(* Logix 5000 project; controller cal1615 1756-L62 rev 20.11; software revision 20.05; part 13 of 81 *)
(* tags used below, declared in another part *)
   FAULT : BOOL;   // Fault AFI
   p01_ai_prs : REAL;   // System Inputs Oxidizer Differential Pressure
   p01_ai_tc : REAL;   // System Inputs Oxidizer Inlet Temperature
   p01_int_from_oxidizer : INT[10];   // System Oxidizer Int from Oxidizer
   p01_int_to_oxidizer : INT;   // System Oxidizer Int to Oxidizer
   p01_param_tension_deviation : REAL;
   p01r01 : routine;
   p01r03_oxidizer_prs : SYS_SCP;   // System Inputs Oxidizer Differential Pressure Scaling
   p01r03_prs_input_max : REAL;
   p01r03_prs_input_min : REAL;
   p01r03_prs_output_max : REAL;
   p01r03_prs_output_min : REAL;
   p01r09_pb_global_reset : BOOL;   // System Modes PB: Global Fault Reset
   p01r12_master_ramped_speed : REAL;   // System Line Accel Decel Control Master Ramped Speed
   p01r12_selected_line_speed : REAL;   // System Line Accel Decel Control Selected Line Speed
   p01r13 : routine;   // System Line Start Sequence
   p01r13_check_status : BOOL;   // System Line Start Sequence Check Status
   p01r13_check_status_time : REAL;   // System Line Start Sequence Check Status
   p01r13_check_status_timer : TIMER;   // System Line Start Sequence Check Status Timer
   p01r13_check_tension : TIMER;   // System Line Start Sequence Check Tension
   p01r13_letoff_tension_ok : BOOL;   // System Line Start Sequence Letoff Tension Ok
   p01r13_line_running : BOOL;   // System Line Start Sequence Line Running
   p01r13_line_slow_ramp : BOOL;   // System Line Start Sequence Start Line to Slow Speed
   p01r13_line_start : SYS_ENC;   // System Line Start Sequence Encoder
   p01r13_permissive_drives : BOOL;   // System Line Start Sequence Permissive Drives
   p01r13_permissive_line_run : BOOL;   // System Line Start Sequence Permissive Line Run
   p01r13_permissive_oven : BOOL;   // System Line start Sequence Permissive Ovens
   p01r13_request_run : BOOL;   // System Line Start Sequence Request Run
   p01r13_request_stop : BOOL;   // System Line Start Sequence Request Stop
   p01r13_state : DINT;   // System Line Start Sequence Sequencer Step
   p01r13_status : DINT;   // System Line Start Sequence Encoded Step
   p01r13_tension_ok : BOOL;   // System Line Start Sequence Slow Speed Tension Ok
   p01r13_timer_fault : TIMER[8];   // System Line Start Sequence Fault Dwell Timer
   p01r13_timer_line_start_warning_dwell : TIMER;   // System Line Start Sequence Pre Start Warning Dwell Timer
   p01r13_timer_line_stop_dwell : TIMER;   // System Line Start Sequence Line Stop Dwell Timer
   p01r13_timer_switch_to_stretch_dwell : TIMER;   // System Line Start Sequence Setpoint Stretch to Tension Dwell Timer
   p01r13_timer_warning : TIMER[8];   // System Line Start Sequence Warning Dwell Timer
   p01r13_ts1_tension_ok : BOOL;   // System Line Start Sequence TS 1 Tension Ok
   p01r13_ts2_tension_ok : BOOL;   // System Line Start Sequence TS 2 Tension Ok
   p01r13_winder_tension_ok : BOOL;   // System Line Start Sequence Winder Tension Ok
   p01r14 : routine;
   p01r14_msg_read : MESSAGE;   // System Oxidizer Message Read
   p01r14_msg_read_retry_timer : TIMER;
   p01r14_msg_read_timer : TIMER;   // System Oxidizer Read Dwell
   p01r14_msg_write : MESSAGE;   // System Oxidizer Message Write
   p01r14_msg_write_retry_timer : TIMER;   // System Oxidizer Message Retry Timer
   p01r14_msg_write_timer : TIMER;   // System Oxidizer Message Read Dwell
   p01r14_oxidizer_heart_beat_off : TIMER;   // System Oxidizer Heart Beat Off Timer
   p01r14_oxidizer_heart_beat_ok : BOOL;   // System Oxidizer Heart Beat Ok
   p01r14_oxidizer_heart_beat_on : TIMER;   // System Oxidizer Heart Beat On Timer
   p01r14_oxidizer_mass_flow : REAL;   // System Oxidizer Oxidizer Mass Flow [SCFM]
   p01r14_timer_fault : TIMER[10];   // System Oxidizer Fault Dwell Timer
   p01r14_timer_warning : TIMER[5];
   p11r02_shutdown_temp : BOOL;   // Zone 1 Misc Control Safe Shutdown Temperature
   p11r20_state : DINT;   // Zone 1 Temperature Control State
   p11r30_request_heat : BOOL;   // Zone 1 Temperature Control Request Heat
   p12r02_shutdown_temp : BOOL;   // Zone 2 Misc Control Safe Shutdown Temperature
   p12r20_state : DINT;   // Zone 2 Temperature Control State
   p12r30_request_heat : BOOL;   // Zone 2 Temperature Control Request Heat
   p13r02_shutdown_temp : BOOL;   // Zone 3 Misc Control Safe Shutdown Temperature
   p13r20_state : DINT;   // Zone 3 Temperature Control State
   p13r30_request_cool : BOOL;   // Zone 3 Temperature Control Request Cooling
   p20_di_acc_empty : BOOL;   // Letoff Digital Input Letoff Accumulator Empty Position
   p20r10_pid_tens : PID;   // Letoff Letoff Speed Control Tension PID
   p22r10_pid_psn : PID;   // Tension Stand 1 Speed Tension PID Dancer Position
   p25r10_pid_psn : PID;   // Tension Stand 2 Speed Tension PID Dancer Position Process Variable
   p29r10_tension_error : REAL;   // Winder Winder A Tension Error winder_tension_sp - Load Cell [lbf]
(* P01_System, continued *)

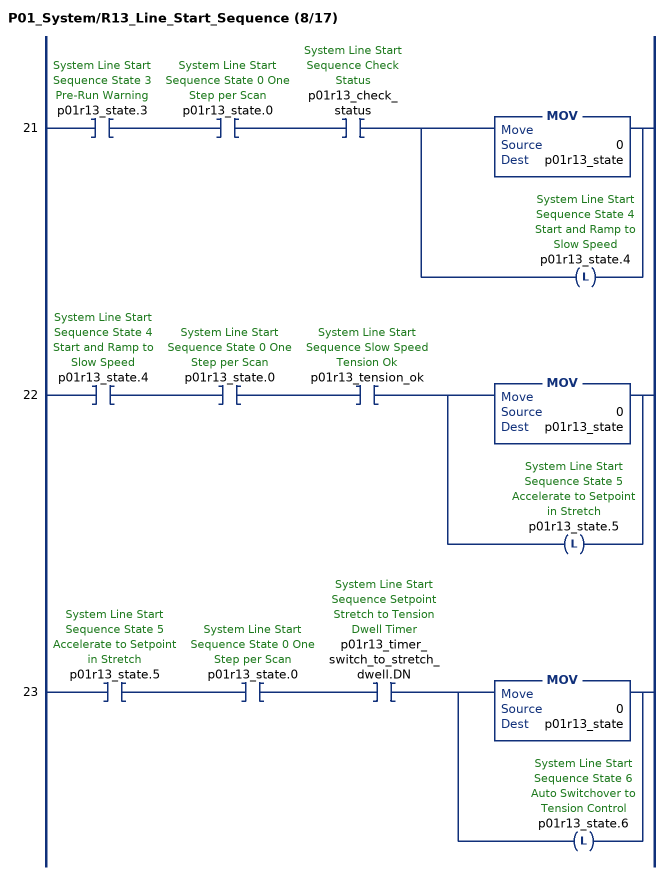
   [picture p162: P01_System/R13_Line_Start_Sequence rungs 21-23]
   21: XIC(p01r13_state.3)XIC(p01r13_state.0)XIC(p01r13_check_status)[MOV(0,p01r13_state) ,OTL(p01r13_state.4) ];
   22: XIC(p01r13_state.4)XIC(p01r13_state.0)XIC(p01r13_tension_ok)[MOV(0,p01r13_state) ,OTL(p01r13_state.5) ];
   23: XIC(p01r13_state.5)XIC(p01r13_state.0)XIC(p01r13_timer_switch_to_stretch_dwell.DN)[MOV(0,p01r13_state) ,OTL(p01r13_state.6) ];
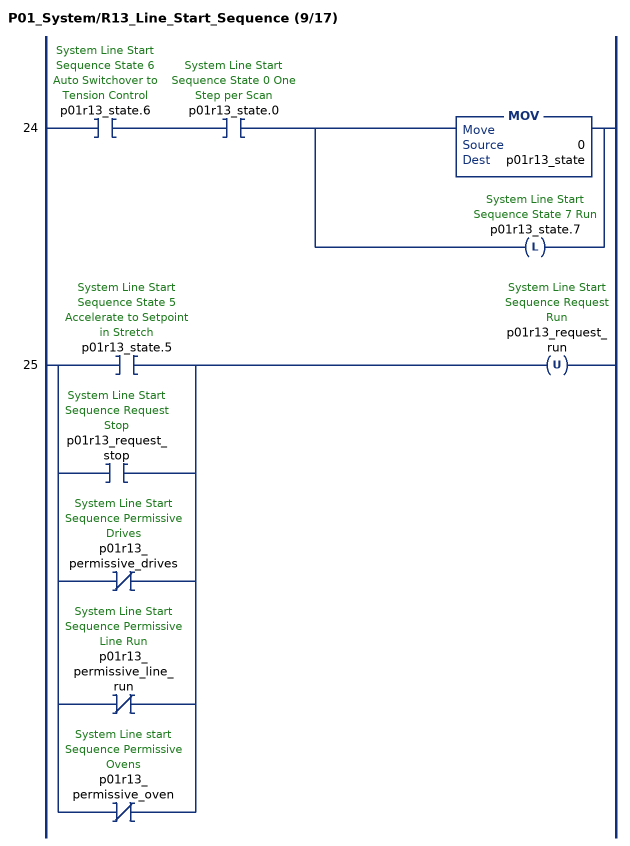
   24: XIC(p01r13_state.6)XIC(p01r13_state.0)[MOV(0,p01r13_state) ,OTL(p01r13_state.7) ];
   25: [XIC(p01r13_state.5) ,XIC(p01r13_request_stop) ,XIO(p01r13_permissive_drives) ,XIO(p01r13_permissive_line_run) ,XIO(p01r13_permissive_oven) ]OTU(p01r13_request_run);
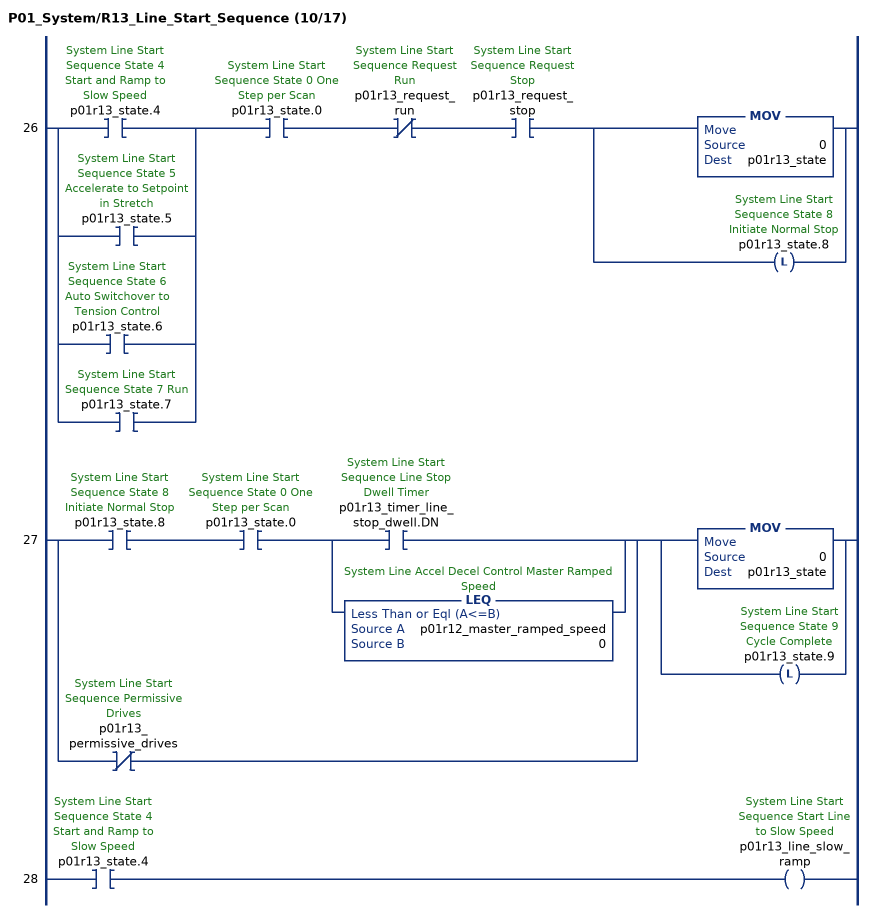
   26: [XIC(p01r13_state.4) ,XIC(p01r13_state.5) ,XIC(p01r13_state.6) ,XIC(p01r13_state.7) ]XIC(p01r13_state.0)XIO(p01r13_request_run)XIC(p01r13_request_stop)[MOV(0,p01r13_state) ,OTL(p01r13_state.8) ];
   27: [XIC(p01r13_state.8) XIC(p01r13_state.0) [XIC(p01r13_timer_line_stop_dwell.DN) ,LEQ(p01r12_master_ramped_speed,0) ] ,XIO(p01r13_permissive_drives) ][MOV(0,p01r13_state) ,OTL(p01r13_state.9) ];
   28: XIC(p01r13_state.4)OTE(p01r13_line_slow_ramp);
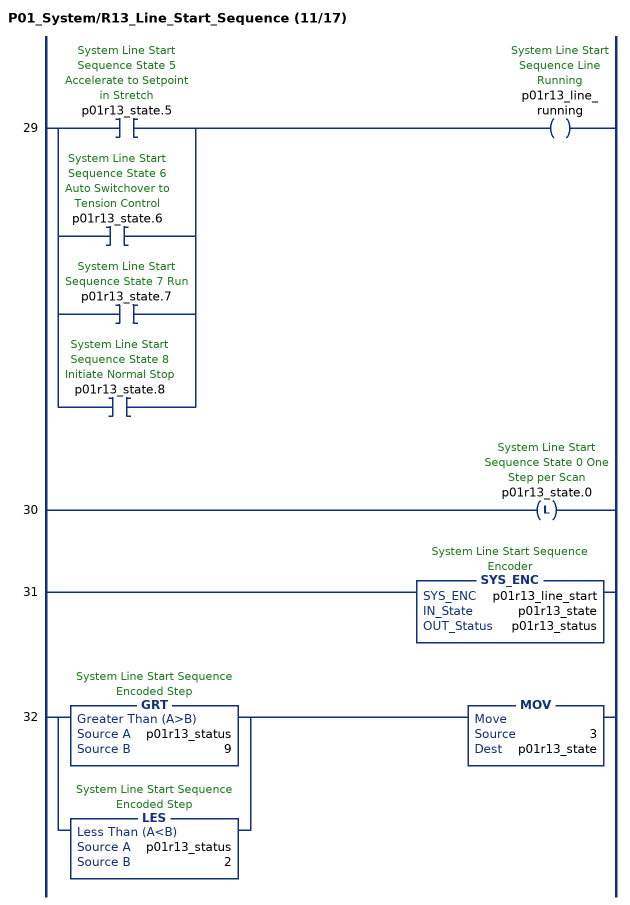
   29: [XIC(p01r13_state.5) ,XIC(p01r13_state.6) ,XIC(p01r13_state.7) ,XIC(p01r13_state.8) ]OTE(p01r13_line_running);
   30: OTL(p01r13_state.0);
   31: SYS_ENC(p01r13_line_start,p01r13_state,p01r13_status);
   32: [GRT(p01r13_status,9) ,LES(p01r13_status,2) ]MOV(3,p01r13_state);
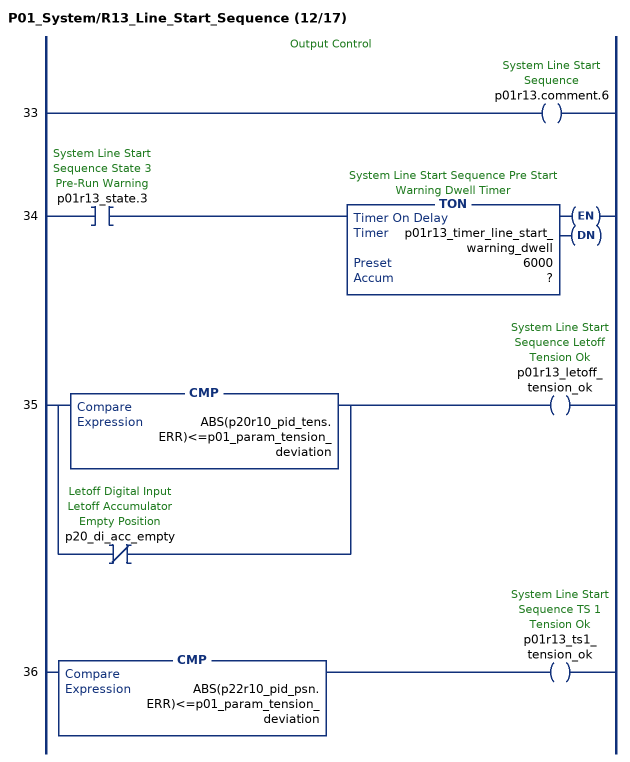
   // Output Control
   33: OTE(p01r13.comment.6);
   34: XIC(p01r13_state.3)TON(p01r13_timer_line_start_warning_dwell,?,?);
   35: [CMP(ABS(p20r10_pid_tens.ERR)<=p01_param_tension_deviation) ,XIO(p20_di_acc_empty) ]OTE(p01r13_letoff_tension_ok);
   36: CMP(ABS(p22r10_pid_psn.ERR)<=p01_param_tension_deviation)OTE(p01r13_ts1_tension_ok);
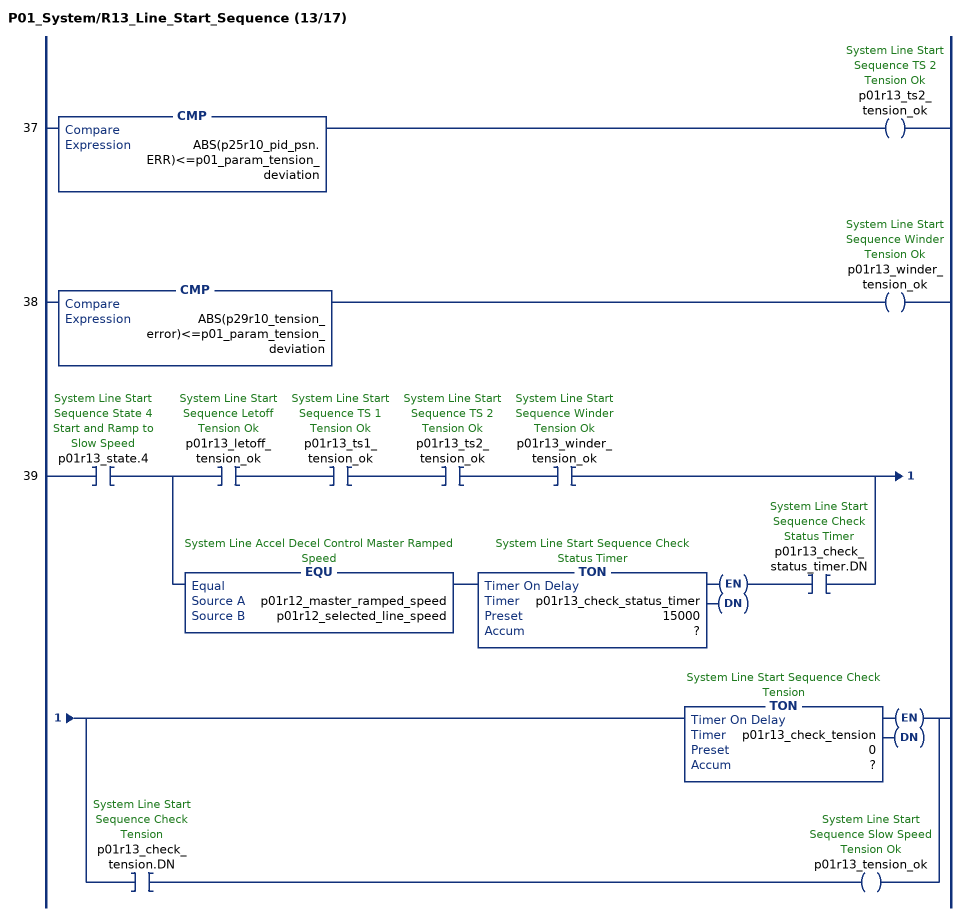
   37: CMP(ABS(p25r10_pid_psn.ERR)<=p01_param_tension_deviation)OTE(p01r13_ts2_tension_ok);
   38: CMP(ABS(p29r10_tension_error)<=p01_param_tension_deviation)OTE(p01r13_winder_tension_ok);
   39: XIC(p01r13_state.4)[XIC(p01r13_letoff_tension_ok) XIC(p01r13_ts1_tension_ok) XIC(p01r13_ts2_tension_ok) XIC(p01r13_winder_tension_ok) ,EQU(p01r12_master_ramped_speed,p01r12_selected_line_speed) TON(p01r13_check_status_timer,?,?) XIC(p01r13_check_status_timer.DN) ][TON(p01r13_check_tension,?,?) ,XIC(p01r13_check_tension.DN) OTE(p01r13_tension_ok) ];
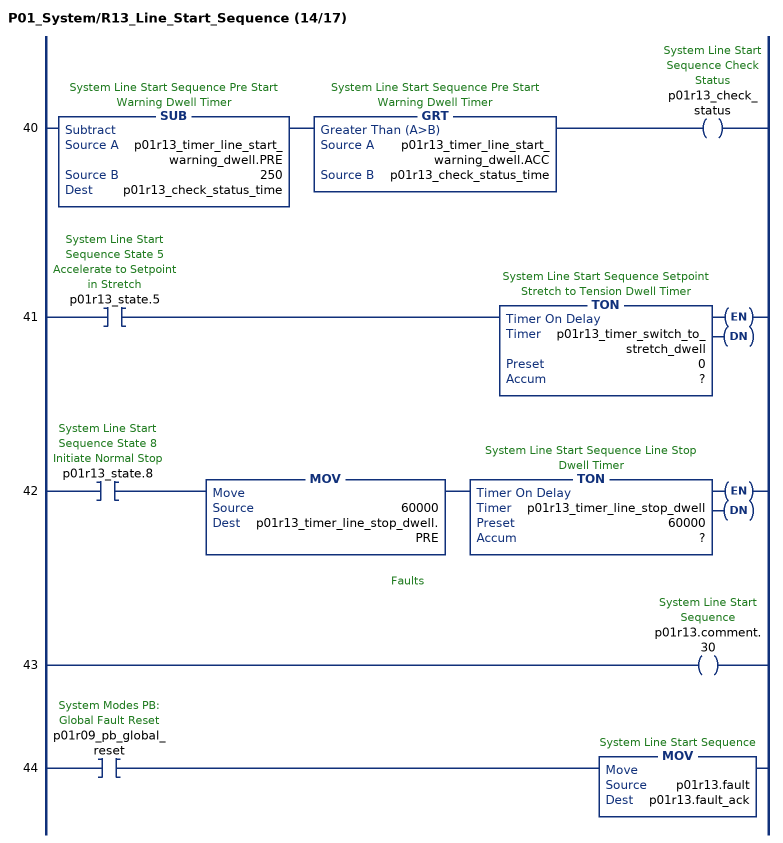
   40: SUB(p01r13_timer_line_start_warning_dwell.PRE,250,p01r13_check_status_time)GRT(p01r13_timer_line_start_warning_dwell.ACC,p01r13_check_status_time)OTE(p01r13_check_status);
   41: XIC(p01r13_state.5)TON(p01r13_timer_switch_to_stretch_dwell,?,?);
   42: XIC(p01r13_state.8)MOV(60000,p01r13_timer_line_stop_dwell.PRE)TON(p01r13_timer_line_stop_dwell,?,?);
   // Faults
   43: OTE(p01r13.comment.30);
   44: XIC(p01r09_pb_global_reset)MOV(p01r13.fault,p01r13.fault_ack);
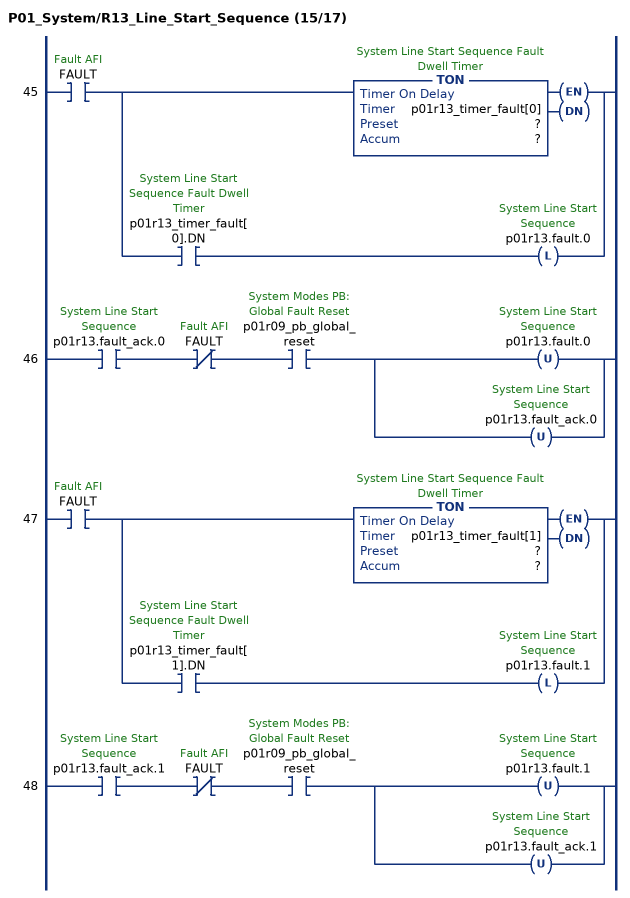
   45: XIC(FAULT)[TON(p01r13_timer_fault[0],?,?) ,XIC(p01r13_timer_fault[0].DN) OTL(p01r13.fault.0) ];
   46: XIC(p01r13.fault_ack.0)XIO(FAULT)XIC(p01r09_pb_global_reset)[OTU(p01r13.fault.0) ,OTU(p01r13.fault_ack.0) ];
   47: XIC(FAULT)[TON(p01r13_timer_fault[1],?,?) ,XIC(p01r13_timer_fault[1].DN) OTL(p01r13.fault.1) ];
   48: XIC(p01r13.fault_ack.1)XIO(FAULT)XIC(p01r09_pb_global_reset)[OTU(p01r13.fault.1) ,OTU(p01r13.fault_ack.1) ];
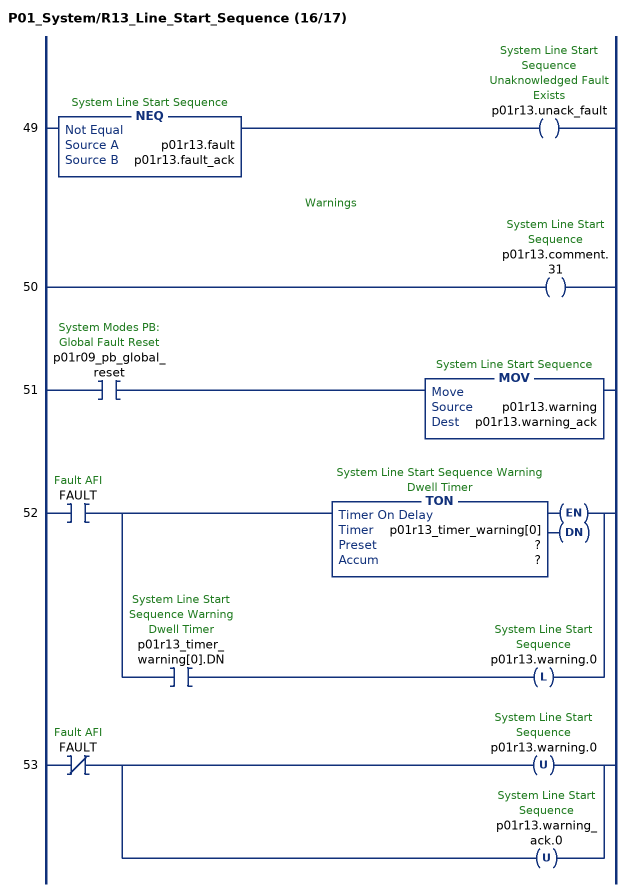
   49: NEQ(p01r13.fault,p01r13.fault_ack)OTE(p01r13.unack_fault);
   // Warnings
   50: OTE(p01r13.comment.31);
   51: XIC(p01r09_pb_global_reset)MOV(p01r13.warning,p01r13.warning_ack);
   52: XIC(FAULT)[TON(p01r13_timer_warning[0],?,?) ,XIC(p01r13_timer_warning[0].DN) OTL(p01r13.warning.0) ];
   53: XIO(FAULT)[OTU(p01r13.warning.0) ,OTU(p01r13.warning_ack.0) ];
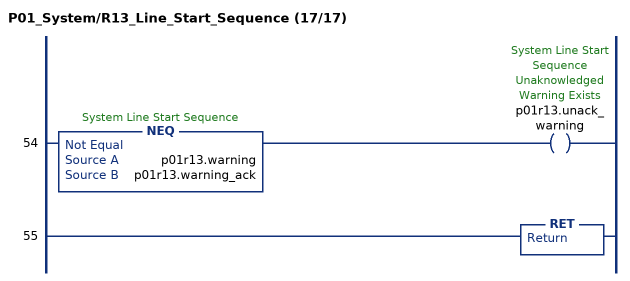
   54: NEQ(p01r13.warning,p01r13.warning_ack)OTE(p01r13.unack_warning);
   55: RET();
END_ROUTINE

ROUTINE R14_Oxidizer   (* ladder *)
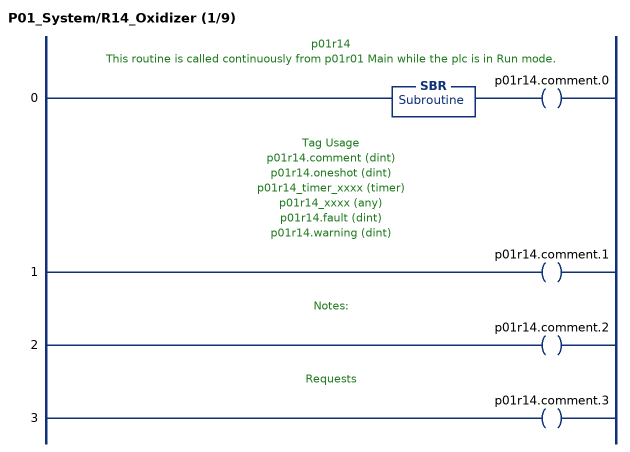
   // p01r14
   // This routine is called continuously from p01r01 Main while the plc is in Run mode.
   0: SBR()OTE(p01r14.comment.0);
   // Tag Usage
   // p01r14.comment (dint)
   // p01r14.oneshot (dint)
   // p01r14_timer_xxxx (timer)
   // p01r14_xxxx (any)
   // p01r14.fault (dint)
   // p01r14.warning (dint)
   1: OTE(p01r14.comment.1);
   // Notes:
   2: OTE(p01r14.comment.2);
   // Requests
   3: OTE(p01r14.comment.3);
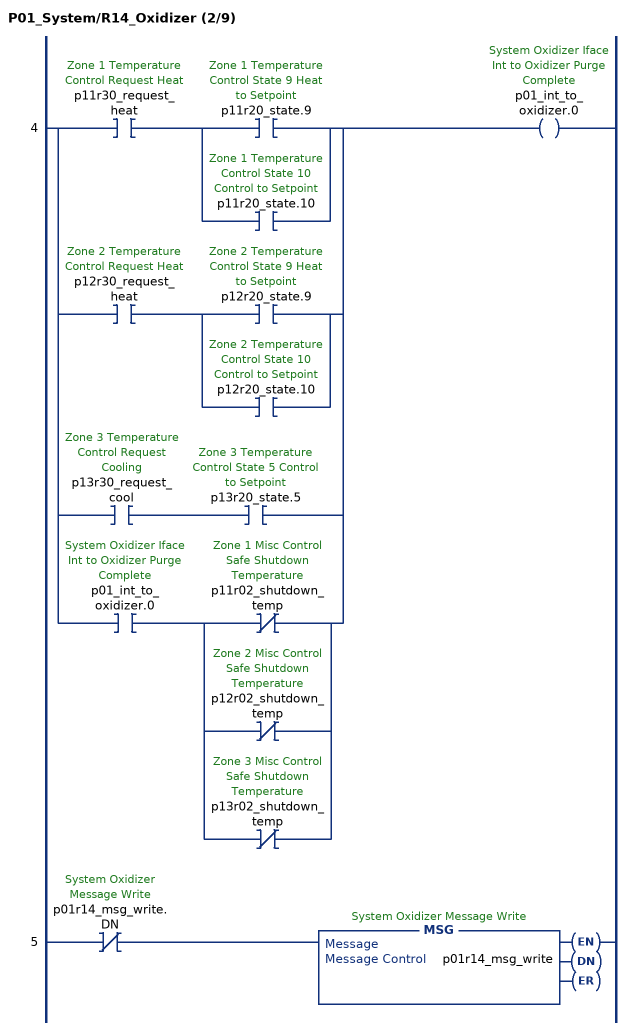
   4: [XIC(p11r30_request_heat) [XIC(p11r20_state.9) ,XIC(p11r20_state.10) ] ,XIC(p12r30_request_heat) [XIC(p12r20_state.9) ,XIC(p12r20_state.10) ] ,XIC(p13r30_request_cool) XIC(p13r20_state.5) ,XIC(p01_int_to_oxidizer.0) [XIO(p11r02_shutdown_temp) ,XIO(p12r02_shutdown_temp) ,XIO(p13r02_shutdown_temp) ] ]OTE(p01_int_to_oxidizer.0);
   5: XIO(p01r14_msg_write.DN)MSG(p01r14_msg_write);
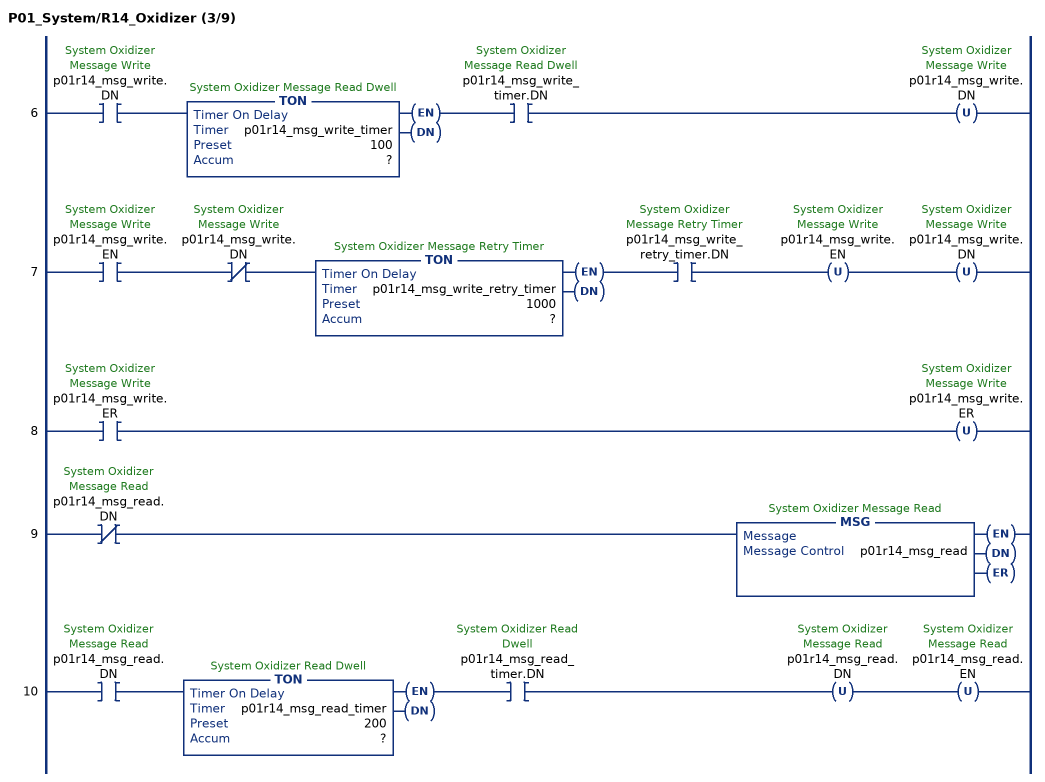
   6: XIC(p01r14_msg_write.DN)TON(p01r14_msg_write_timer,?,?)XIC(p01r14_msg_write_timer.DN)OTU(p01r14_msg_write.DN);
   7: XIC(p01r14_msg_write.EN)XIO(p01r14_msg_write.DN)TON(p01r14_msg_write_retry_timer,?,?)XIC(p01r14_msg_write_retry_timer.DN)OTU(p01r14_msg_write.EN)OTU(p01r14_msg_write.DN);
   8: XIC(p01r14_msg_write.ER)OTU(p01r14_msg_write.ER);
   9: XIO(p01r14_msg_read.DN)MSG(p01r14_msg_read);
   10: XIC(p01r14_msg_read.DN)TON(p01r14_msg_read_timer,?,?)XIC(p01r14_msg_read_timer.DN)OTU(p01r14_msg_read.DN)OTU(p01r14_msg_read.EN);
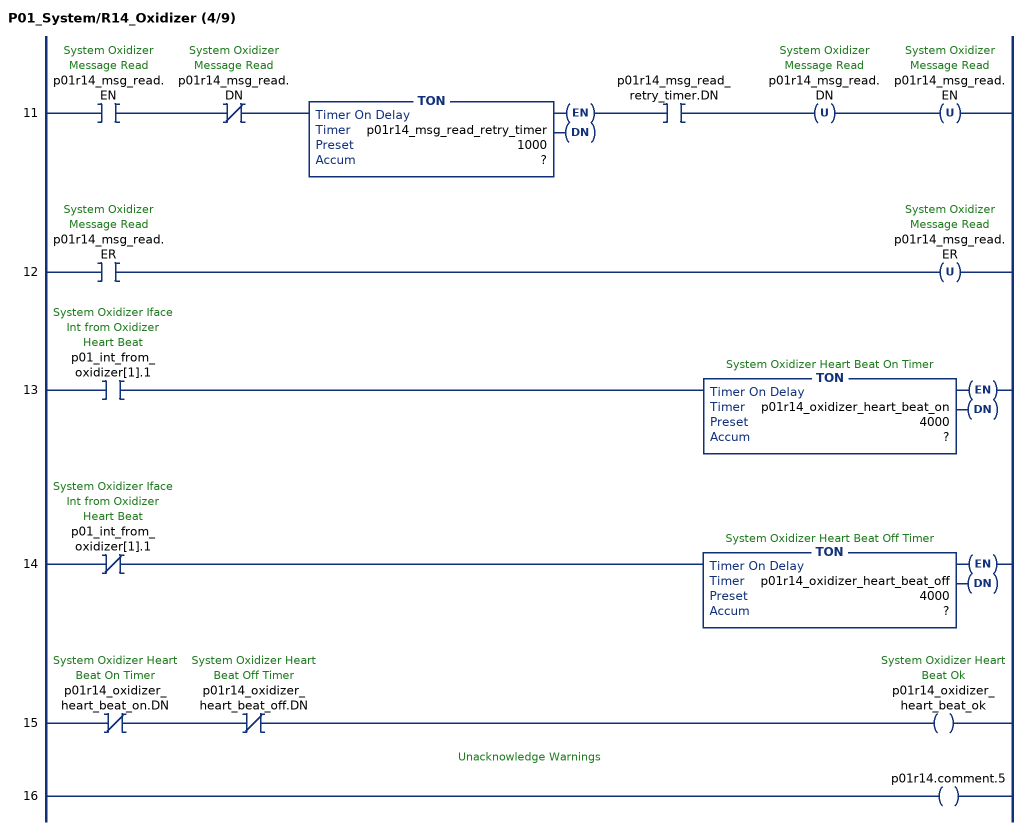
   11: XIC(p01r14_msg_read.EN)XIO(p01r14_msg_read.DN)TON(p01r14_msg_read_retry_timer,?,?)XIC(p01r14_msg_read_retry_timer.DN)OTU(p01r14_msg_read.DN)OTU(p01r14_msg_read.EN);
   12: XIC(p01r14_msg_read.ER)OTU(p01r14_msg_read.ER);
   13: XIC(p01_int_from_oxidizer[1].1)TON(p01r14_oxidizer_heart_beat_on,?,?);
   14: XIO(p01_int_from_oxidizer[1].1)TON(p01r14_oxidizer_heart_beat_off,?,?);
   15: XIO(p01r14_oxidizer_heart_beat_on.DN)XIO(p01r14_oxidizer_heart_beat_off.DN)OTE(p01r14_oxidizer_heart_beat_ok);
   // Unacknowledge Warnings
   16: OTE(p01r14.comment.5);
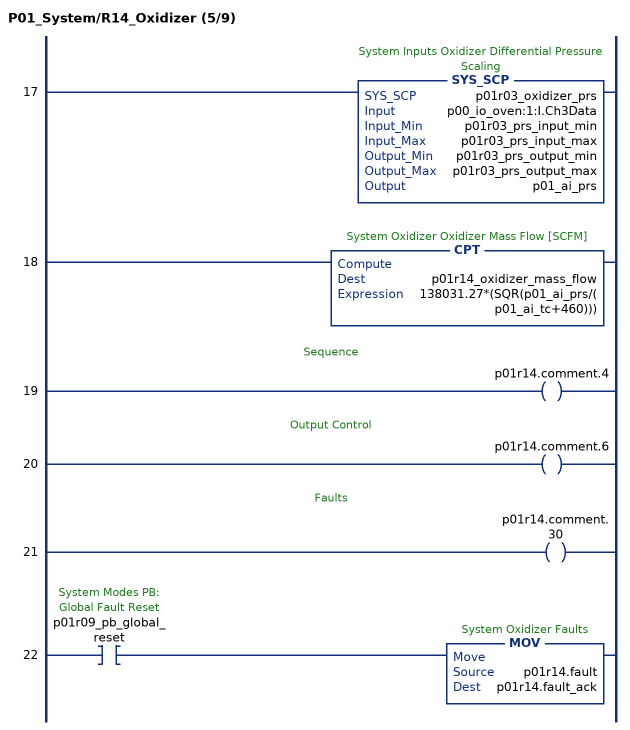
   17: SYS_SCP(p01r03_oxidizer_prs,p00_io_oven:1:I.Ch3Data,p01r03_prs_input_min,p01r03_prs_input_max,p01r03_prs_output_min,p01r03_prs_output_max,p01_ai_prs);
   18: CPT(p01r14_oxidizer_mass_flow,138031.27*(SQR(p01_ai_prs/(p01_ai_tc+460))));
   // Sequence
   19: OTE(p01r14.comment.4);
   // Output Control
   20: OTE(p01r14.comment.6);
   // Faults
   21: OTE(p01r14.comment.30);
   22: XIC(p01r09_pb_global_reset)MOV(p01r14.fault,p01r14.fault_ack);
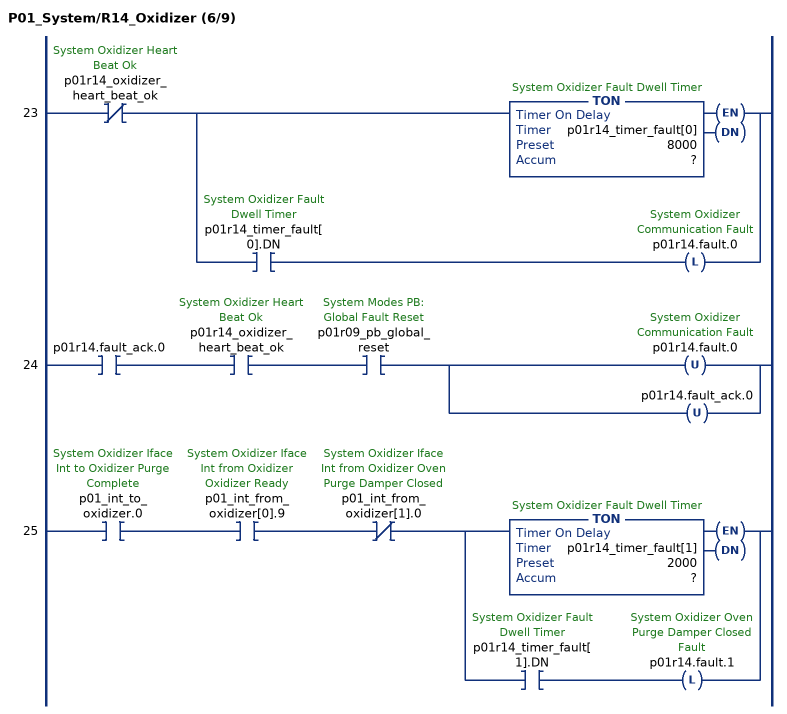
   23: XIO(p01r14_oxidizer_heart_beat_ok)[TON(p01r14_timer_fault[0],?,?) ,XIC(p01r14_timer_fault[0].DN) OTL(p01r14.fault.0) ];
   24: XIC(p01r14.fault_ack.0)XIC(p01r14_oxidizer_heart_beat_ok)XIC(p01r09_pb_global_reset)[OTU(p01r14.fault.0) ,OTU(p01r14.fault_ack.0) ];
   25: XIC(p01_int_to_oxidizer.0)XIC(p01_int_from_oxidizer[0].9)XIO(p01_int_from_oxidizer[1].0)[TON(p01r14_timer_fault[1],?,?) ,XIC(p01r14_timer_fault[1].DN) OTL(p01r14.fault.1) ];
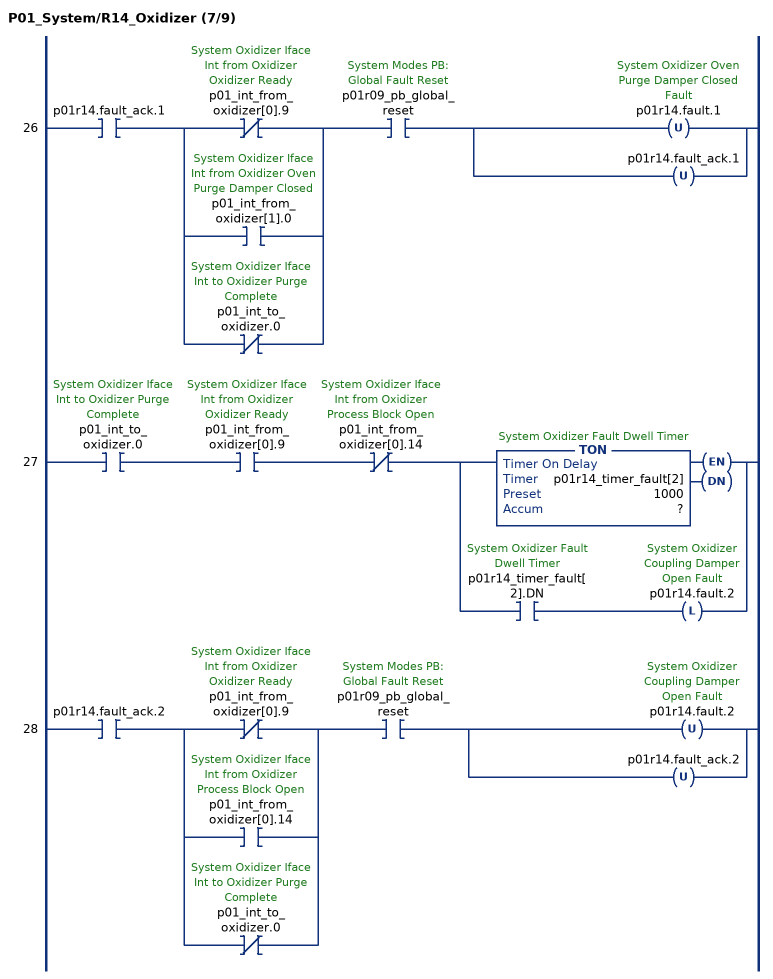
   26: XIC(p01r14.fault_ack.1)[XIO(p01_int_from_oxidizer[0].9) ,XIC(p01_int_from_oxidizer[1].0) ,XIO(p01_int_to_oxidizer.0) ]XIC(p01r09_pb_global_reset)[OTU(p01r14.fault.1) ,OTU(p01r14.fault_ack.1) ];
   27: XIC(p01_int_to_oxidizer.0)XIC(p01_int_from_oxidizer[0].9)XIO(p01_int_from_oxidizer[0].14)[TON(p01r14_timer_fault[2],?,?) ,XIC(p01r14_timer_fault[2].DN) OTL(p01r14.fault.2) ];
   28: XIC(p01r14.fault_ack.2)[XIO(p01_int_from_oxidizer[0].9) ,XIC(p01_int_from_oxidizer[0].14) ,XIO(p01_int_to_oxidizer.0) ]XIC(p01r09_pb_global_reset)[OTU(p01r14.fault.2) ,OTU(p01r14.fault_ack.2) ];
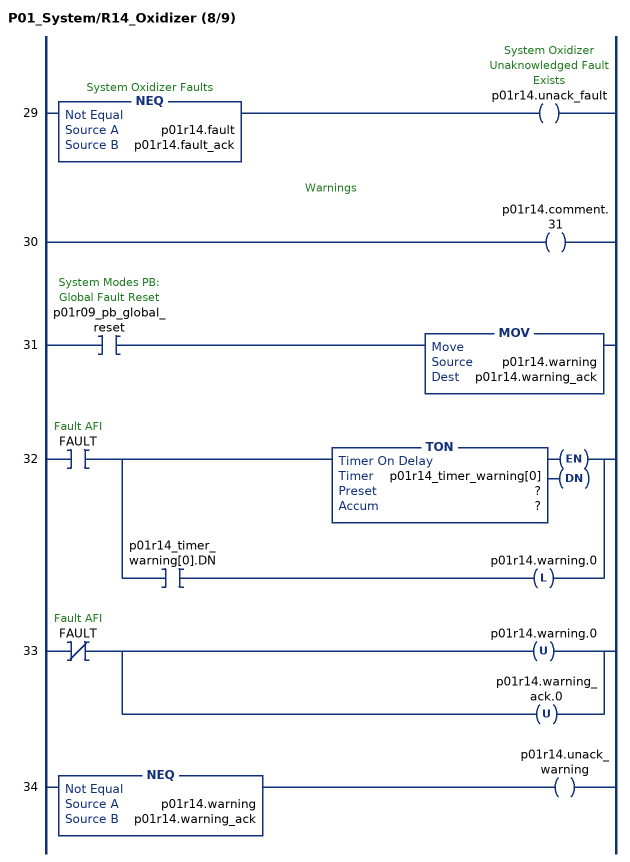
   29: NEQ(p01r14.fault,p01r14.fault_ack)OTE(p01r14.unack_fault);
   // Warnings
   30: OTE(p01r14.comment.31);
   31: XIC(p01r09_pb_global_reset)MOV(p01r14.warning,p01r14.warning_ack);
   32: XIC(FAULT)[TON(p01r14_timer_warning[0],?,?) ,XIC(p01r14_timer_warning[0].DN) OTL(p01r14.warning.0) ];
   33: XIO(FAULT)[OTU(p01r14.warning.0) ,OTU(p01r14.warning_ack.0) ];
   34: NEQ(p01r14.warning,p01r14.warning_ack)OTE(p01r14.unack_warning);
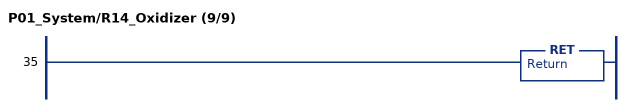
   35: RET();
END_ROUTINE
